// Mitsubishi GX Works2 project: GoodAfterChanges   PLC: FX3G

// global labels: Global1
VAR_GLOBAL
  Start_Day AT X007 : BOOL;
  Output_Analog AT D8282 : INT;
  Check_Input AT M1 : BOOL;
  Work_Day_Light AT Y007 : BOOL;
  End_Day AT M0 : BOOL;
END_VAR
VAR_GLOBAL CONSTANT
  Petel_For_Regular : REAL := 280;
  Lemon_For_Regular : REAL := 455;
END_VAR
VAR_GLOBAL
  Input_Petel AT D2000 : REAL;
  Input_Lemon AT D2002 : REAL;
  Input_Gummy_Bears AT D2004 : REAL;
  Input_Stabilizer AT D2006 : REAL;
  Stock_Petel AT D3000 : REAL;
  Stock_Lemon AT D3002 : REAL;
  Stock_Gummy_Bears AT D3004 : REAL;
  Stock_Stabilizer AT D3006 : REAL;
  Read_Input AT X001 : BOOL;
END_VAR
VAR_GLOBAL CONSTANT
  Petel_For_Special : REAL := 385;
  Lemon_For_Special : REAL := 665;
  Gummy_Bears_For_Special : REAL := 70;
  Stabilizer_For_Special : REAL := 30;
END_VAR
VAR_GLOBAL
  Input_Analog1 AT D8280 : INT;
END_VAR
VAR_GLOBAL CONSTANT
  Normalize : REAL := 404.5;
END_VAR
VAR_GLOBAL
  Type_Ice_Cream AT D4000 : REAL;
END_VAR
VAR_GLOBAL CONSTANT
  Min_Regular : REAL;
  Min_Special : REAL := 6;
  Max_Regular : REAL := 5.0;
END_VAR
VAR_GLOBAL
  Making_Ice_Cream AT Y000 : BOOL;
  Making_Time AT TC1 : BOOL;
  End_Making AT TS1 : BOOL;
  Start_Cooling AT X002 : BOOL;
  Petel_Making AT D4200 : REAL;
  Lemon_Making AT D4202 : REAL;
END_VAR
VAR_GLOBAL CONSTANT
  Total_Petel_Regular : REAL := 350;
  Total_Petel_Special : REAL := 560;
  Total_Lemon_Regular : REAL := 490;
  Total_Lemon_Special : REAL := 700;
END_VAR
VAR_GLOBAL
  Petel_Cooling AT D4204 : REAL;
  Cool_Time AT TC2 : BOOL;
END_VAR
VAR_GLOBAL CONSTANT
  Time_Making_Sec : WORD := 50;
  Time_Cool_Sec : WORD := 80;
END_VAR
VAR_GLOBAL
  Mixing_Pot AT D4208 : REAL;
  Mixing_Reg_Time AT TC3 : BOOL;
  Mixing_Spe_Time AT TC4 : BOOL;
END_VAR
VAR_GLOBAL CONSTANT
  Mixing_Reg_Sec : WORD := 30;
  Mixing_Spe_Sec : WORD := 50;
END_VAR
VAR_GLOBAL
  Regular_Check AT M3 : BOOL;
  Special_Check AT M4 : BOOL;
  Make_Special AT M6 : BOOL;
  Make_Regular AT M5 : BOOL;
  End_Cooling AT TS2 : BOOL;
  Cooling_Ice_Cream AT Y002 : BOOL;
  Temp_Sensor AT X003 : BOOL;
  End_Regular_Mixing AT TS3 : BOOL;
  End_Special_Mixing AT TS4 : BOOL;
  Blink_Helper AT M7 : BOOL;
  Light5 AT Y005 : BOOL;
END_VAR
VAR_GLOBAL CONSTANT
  Blinking_Time : WORD := 5;
END_VAR
VAR_GLOBAL
  Start_Packing AT X004 : BOOL;
  First_Cup AT CC0 : BOOL;
END_VAR
VAR_GLOBAL CONSTANT
  Counter1 : WORD := 1;
END_VAR
VAR_GLOBAL
  Counter_Pack AT CC1 : BOOL;
END_VAR
VAR_GLOBAL CONSTANT
  Counter7 : WORD := 7;
END_VAR
VAR_GLOBAL
  End_Counter1 AT CS0 : BOOL;
  End_Counter7 AT CS1 : BOOL;
  Light4 AT Y004 : BOOL;
  Pack_One AT X000 : BOOL;
  Packs_Amount AT D4400 : REAL;
END_VAR
VAR_GLOBAL CONSTANT
  Add_One : REAL := 1;
END_VAR
VAR_GLOBAL
  Update_Stock AT M2 : BOOL;
END_VAR
VAR_GLOBAL CONSTANT
  Max_Special : REAL := 10.0;
  Gummy_Bears_For_Regular : REAL := 28;
  Stabilizer_For_Regular : REAL := 15;
END_VAR
VAR_GLOBAL
  Lemon_Cooling AT D4206 : REAL;
  Blink5 AT TC5 : BOOL;
  Blink6 AT TC6 : BOOL;
  End_Blink5 AT TS5 : BOOL;
  Light6 AT Y006 : BOOL;
  End_Blink6 AT TS6 : BOOL;
  Emergency_Stop AT X005 : BOOL;
  Finish_Reset AT M8 : BOOL;
END_VAR
VAR_GLOBAL CONSTANT
  Normalize_Back : REAL := 40.45;
END_VAR

// task Task_01 (event TRUE, interval 0, priority 31): POU_01

PROGRAM POU_01
(* structured ladder/FBD written out as ST: instructions are called as NAME(EN, inputs, outputs); _pN, _eN, _tN stand for wires *)
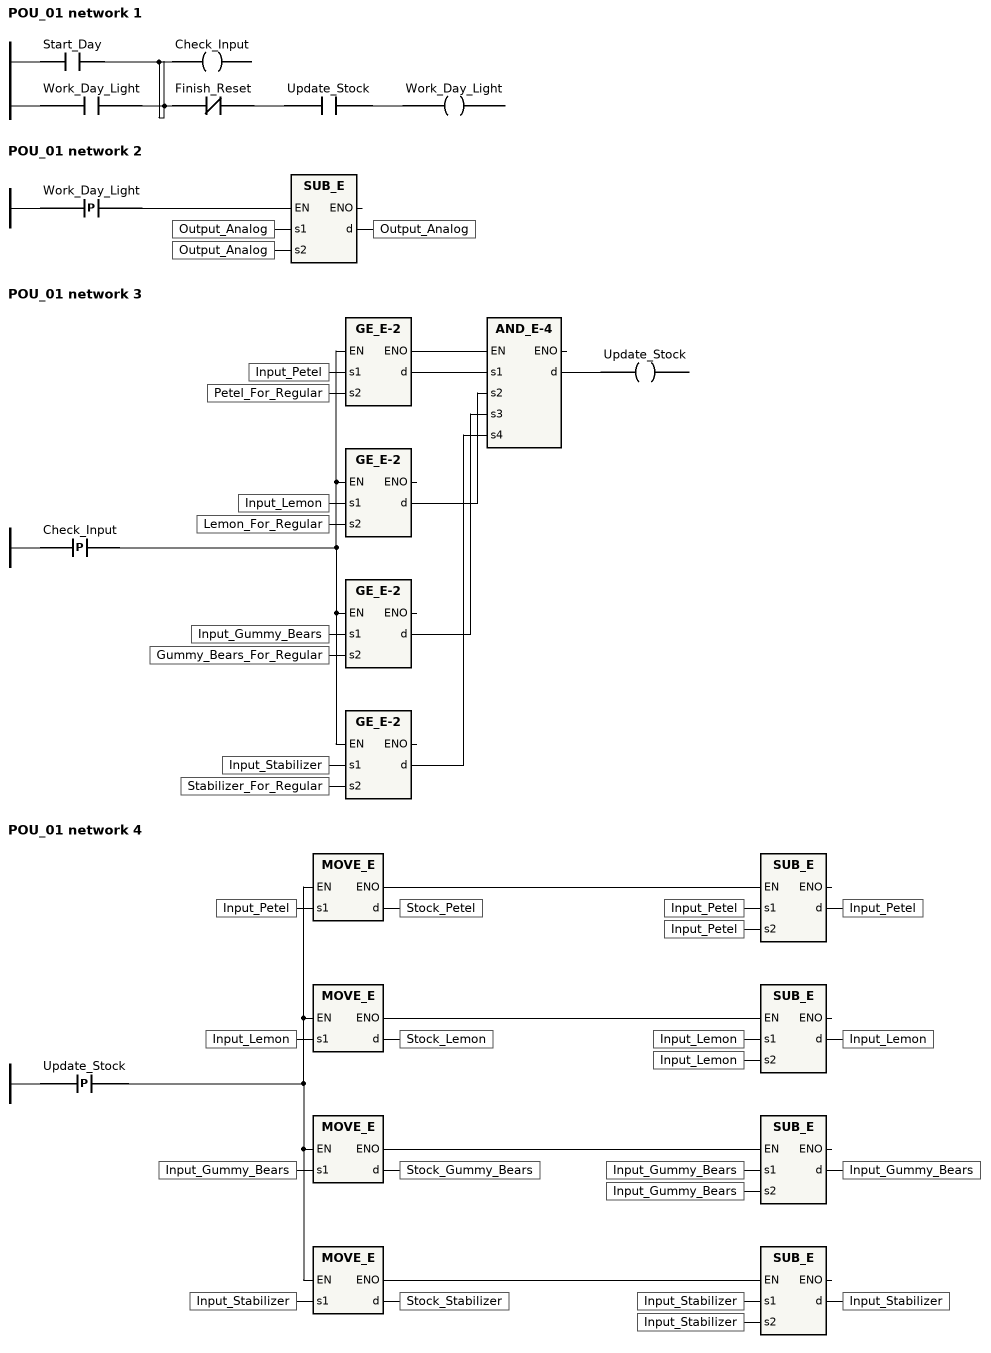
(* network 1 *)
_p1 := Start_Day OR Work_Day_Light;
Check_Input := _p1;
Work_Day_Light := _p1 AND NOT Finish_Reset AND Update_Stock;
(* network 2 *)
SUB_E(LDP(TRUE, Work_Day_Light), Output_Analog, Output_Analog, Output_Analog);
(* network 3 *)
_p1 := LDP(TRUE, Check_Input);
_e3 := GE_E(_p1, Input_Petel, Petel_For_Regular, _t2);
GE_E(_p1, Input_Lemon, Lemon_For_Regular, _t4);
GE_E(_p1, Input_Gummy_Bears, Gummy_Bears_For_Regular, _t5);
GE_E(_p1, Input_Stabilizer, Stabilizer_For_Regular, _t6);
AND_E(_e3, _t2, _t4, _t5, _t6, _t7);
Update_Stock := _t7;
(* network 4 *)
_p1 := LDP(TRUE, Update_Stock);
_e2 := MOVE_E(_p1, Input_Petel, Stock_Petel);
SUB_E(_e2, Input_Petel, Input_Petel, Input_Petel);
_e3 := MOVE_E(_p1, Input_Lemon, Stock_Lemon);
SUB_E(_e3, Input_Lemon, Input_Lemon, Input_Lemon);
_e4 := MOVE_E(_p1, Input_Gummy_Bears, Stock_Gummy_Bears);
SUB_E(_e4, Input_Gummy_Bears, Input_Gummy_Bears, Input_Gummy_Bears);
_e5 := MOVE_E(_p1, Input_Stabilizer, Stock_Stabilizer);
SUB_E(_e5, Input_Stabilizer, Input_Stabilizer, Input_Stabilizer);
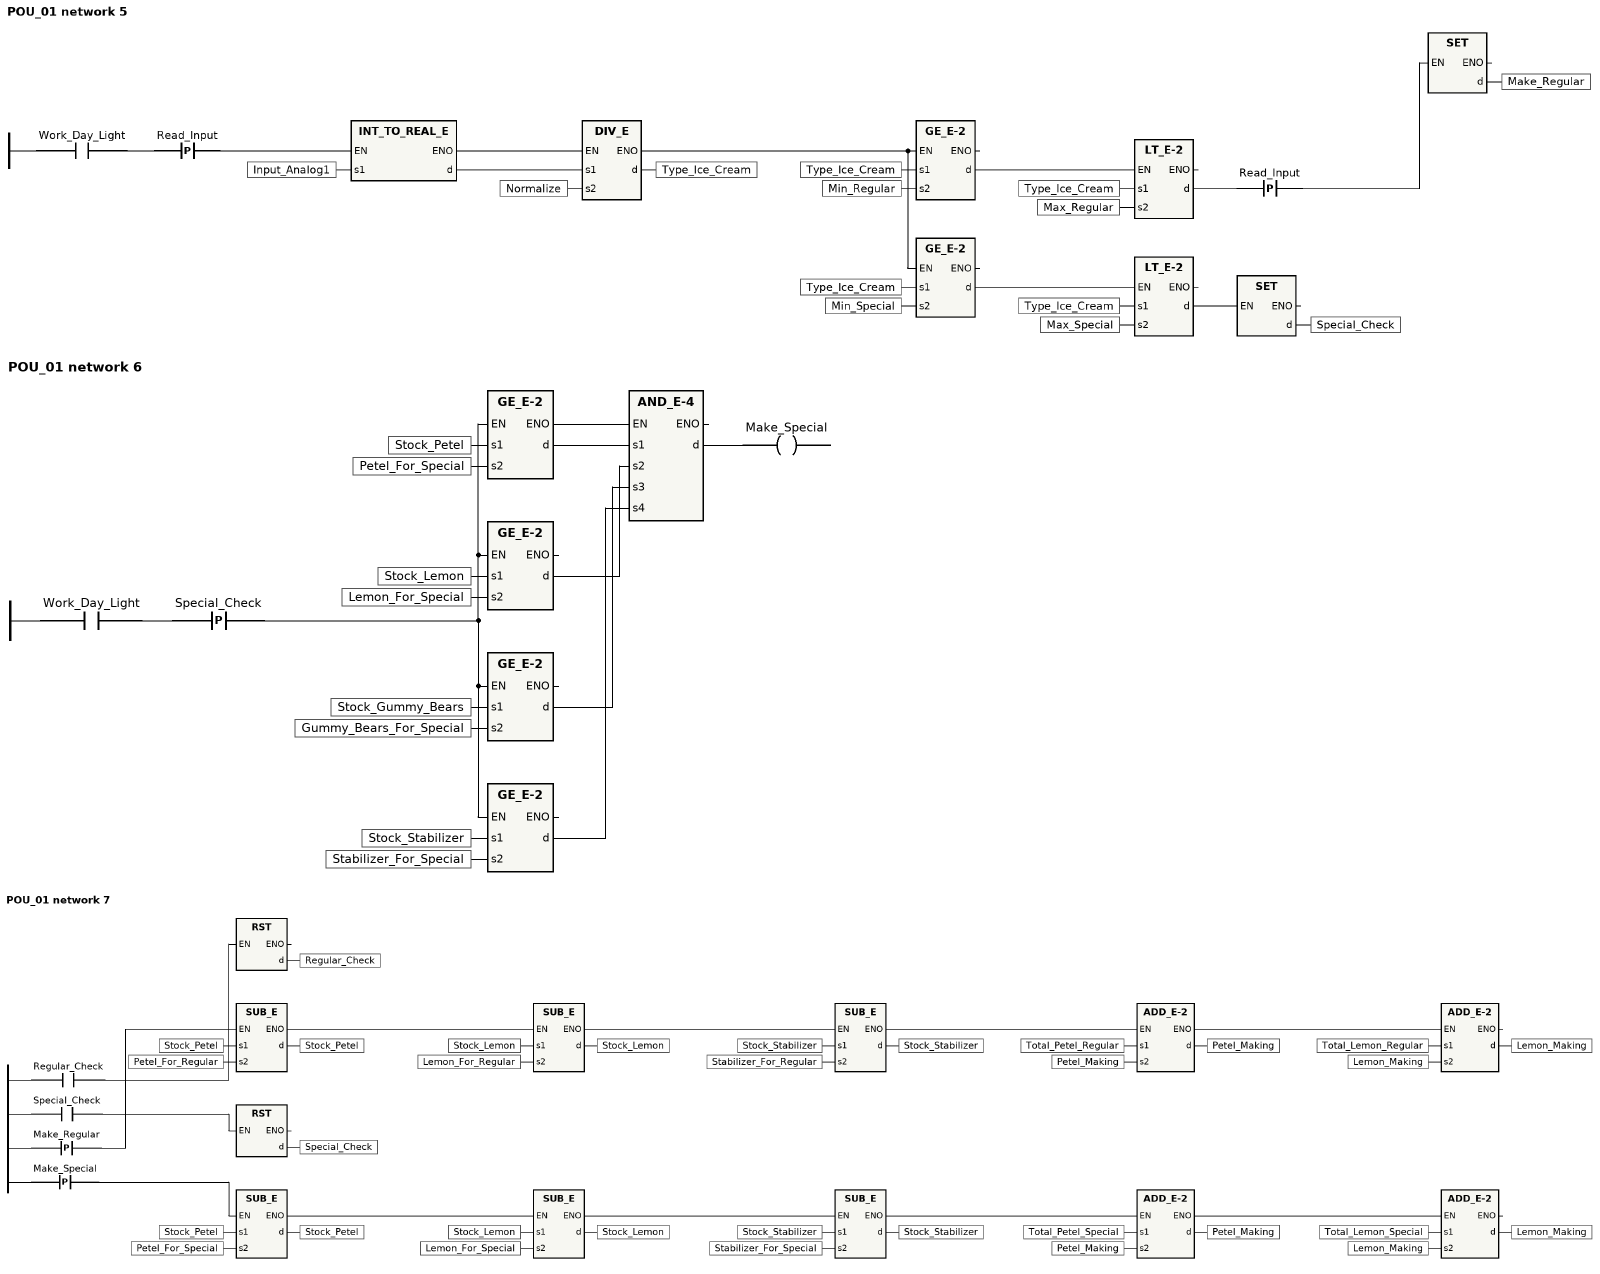
(* network 5 *)
_e2 := INT_TO_REAL_E(Work_Day_Light AND LDP(TRUE, Read_Input), Input_Analog1, _t1);
_e3 := DIV_E(_e2, _t1, Normalize, Type_Ice_Cream);
GE_E(_e3, Type_Ice_Cream, Min_Regular, _t4);
LT_E(_t4, Type_Ice_Cream, Max_Regular, _t5);
SET(_t5 AND LDP(TRUE, Read_Input), Make_Regular);
GE_E(_e3, Type_Ice_Cream, Min_Special, _t6);
LT_E(_t6, Type_Ice_Cream, Max_Special, _t7);
SET(_t7, Special_Check);
(* network 6 *)
_p1 := Work_Day_Light AND LDP(TRUE, Special_Check);
_e3 := GE_E(_p1, Stock_Petel, Petel_For_Special, _t2);
GE_E(_p1, Stock_Lemon, Lemon_For_Special, _t4);
GE_E(_p1, Stock_Gummy_Bears, Gummy_Bears_For_Special, _t5);
GE_E(_p1, Stock_Stabilizer, Stabilizer_For_Special, _t6);
AND_E(_e3, _t2, _t4, _t5, _t6, _t7);
Make_Special := _t7;
(* network 7 *)
RST(Regular_Check, Regular_Check);
RST(Special_Check, Special_Check);
_e1 := SUB_E(LDP(TRUE, Make_Regular), Stock_Petel, Petel_For_Regular, Stock_Petel);
_e2 := SUB_E(_e1, Stock_Lemon, Lemon_For_Regular, Stock_Lemon);
_e3 := SUB_E(_e2, Stock_Stabilizer, Stabilizer_For_Regular, Stock_Stabilizer);
_e4 := ADD_E(_e3, Total_Petel_Regular, Petel_Making, Petel_Making);
ADD_E(_e4, Total_Lemon_Regular, Lemon_Making, Lemon_Making);
_e5 := SUB_E(LDP(TRUE, Make_Special), Stock_Petel, Petel_For_Special, Stock_Petel);
_e6 := SUB_E(_e5, Stock_Lemon, Lemon_For_Special, Stock_Lemon);
_e7 := SUB_E(_e6, Stock_Stabilizer, Stabilizer_For_Special, Stock_Stabilizer);
_e8 := ADD_E(_e7, Total_Petel_Special, Petel_Making, Petel_Making);
ADD_E(_e8, Total_Lemon_Special, Lemon_Making, Lemon_Making);
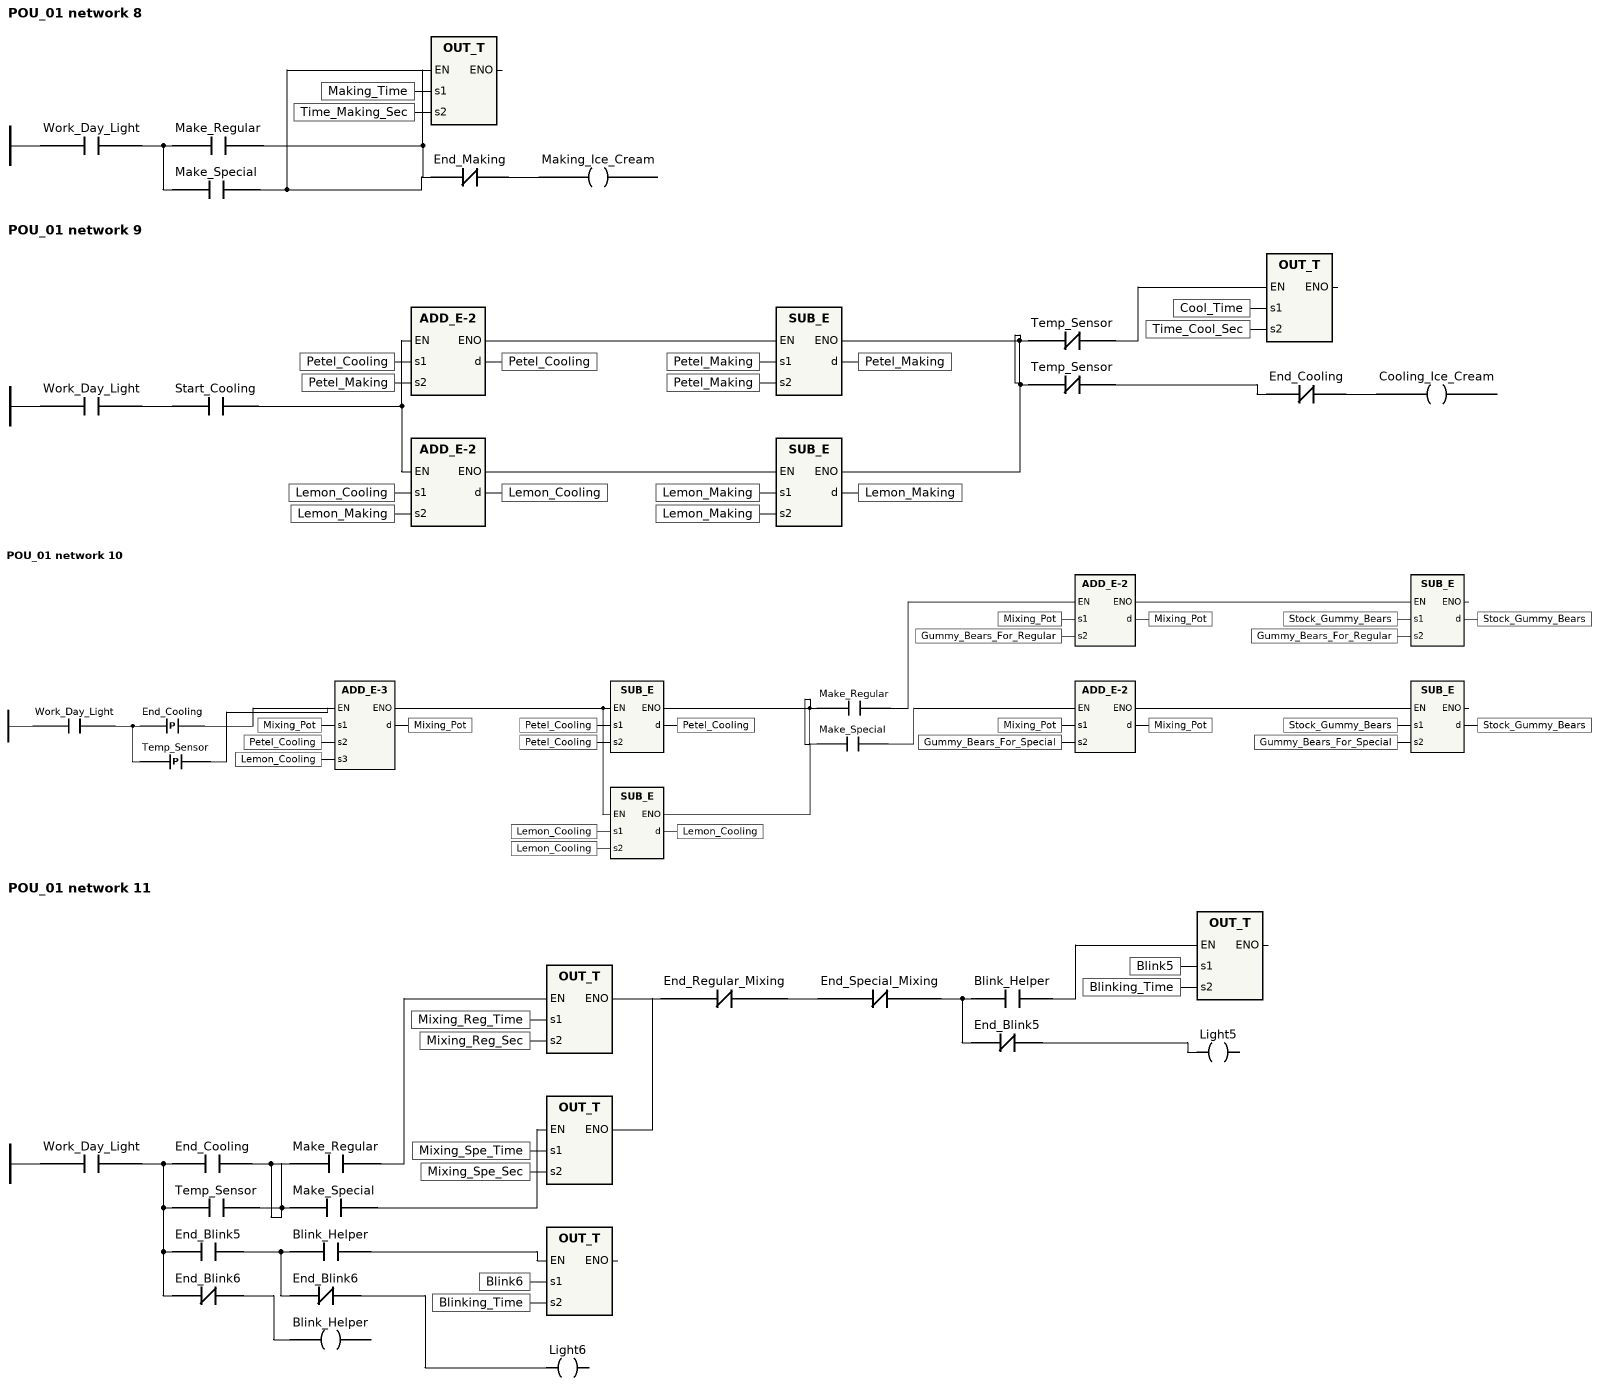
(* network 8 *)
_p1 := (Work_Day_Light AND Make_Regular) OR (Work_Day_Light AND Make_Special);
OUT_T(_p1, Making_Time, Time_Making_Sec);
Making_Ice_Cream := _p1 AND NOT End_Making;
(* network 9 *)
_p1 := Work_Day_Light AND Start_Cooling;
_e2 := ADD_E(_p1, Petel_Cooling, Petel_Making, Petel_Cooling);
_e3 := SUB_E(_e2, Petel_Making, Petel_Making, Petel_Making);
_e4 := ADD_E(_p1, Lemon_Cooling, Lemon_Making, Lemon_Cooling);
_e5 := SUB_E(_e4, Lemon_Making, Lemon_Making, Lemon_Making);
_p6 := _e3 OR _e5;
OUT_T(_p6 AND NOT Temp_Sensor, Cool_Time, Time_Cool_Sec);
Cooling_Ice_Cream := _p6 AND NOT Temp_Sensor AND NOT End_Cooling;
(* network 10 *)
_e1 := ADD_E((Work_Day_Light AND LDP(TRUE, End_Cooling)) OR (Work_Day_Light AND LDP(TRUE, Temp_Sensor)), Mixing_Pot, Petel_Cooling, Lemon_Cooling, Mixing_Pot);
_e2 := SUB_E(_e1, Petel_Cooling, Petel_Cooling, Petel_Cooling);
_e3 := SUB_E(_e1, Lemon_Cooling, Lemon_Cooling, Lemon_Cooling);
_p4 := _e2 OR _e3;
_e5 := ADD_E(_p4 AND Make_Regular, Mixing_Pot, Gummy_Bears_For_Regular, Mixing_Pot);
SUB_E(_e5, Stock_Gummy_Bears, Gummy_Bears_For_Regular, Stock_Gummy_Bears);
_e6 := ADD_E(_p4 AND Make_Special, Mixing_Pot, Gummy_Bears_For_Special, Mixing_Pot);
SUB_E(_e6, Stock_Gummy_Bears, Gummy_Bears_For_Special, Stock_Gummy_Bears);
(* network 11 *)
_p1 := (Work_Day_Light AND End_Cooling) OR (Work_Day_Light AND Temp_Sensor);
_e2 := OUT_T(_p1 AND Make_Regular, Mixing_Reg_Time, Mixing_Reg_Sec);
_e3 := OUT_T(_p1 AND Make_Special, Mixing_Spe_Time, Mixing_Spe_Sec);
_p4 := ((_e2 OR _e3) AND NOT End_Regular_Mixing) AND NOT End_Special_Mixing;
OUT_T(_p4 AND Blink_Helper, Blink5, Blinking_Time);
Light5 := _p4 AND NOT End_Blink5;
_p5 := Work_Day_Light AND End_Blink5;
OUT_T(_p5 AND Blink_Helper, Blink6, Blinking_Time);
Light6 := _p5 AND NOT End_Blink6;
Blink_Helper := Work_Day_Light AND NOT End_Blink6;
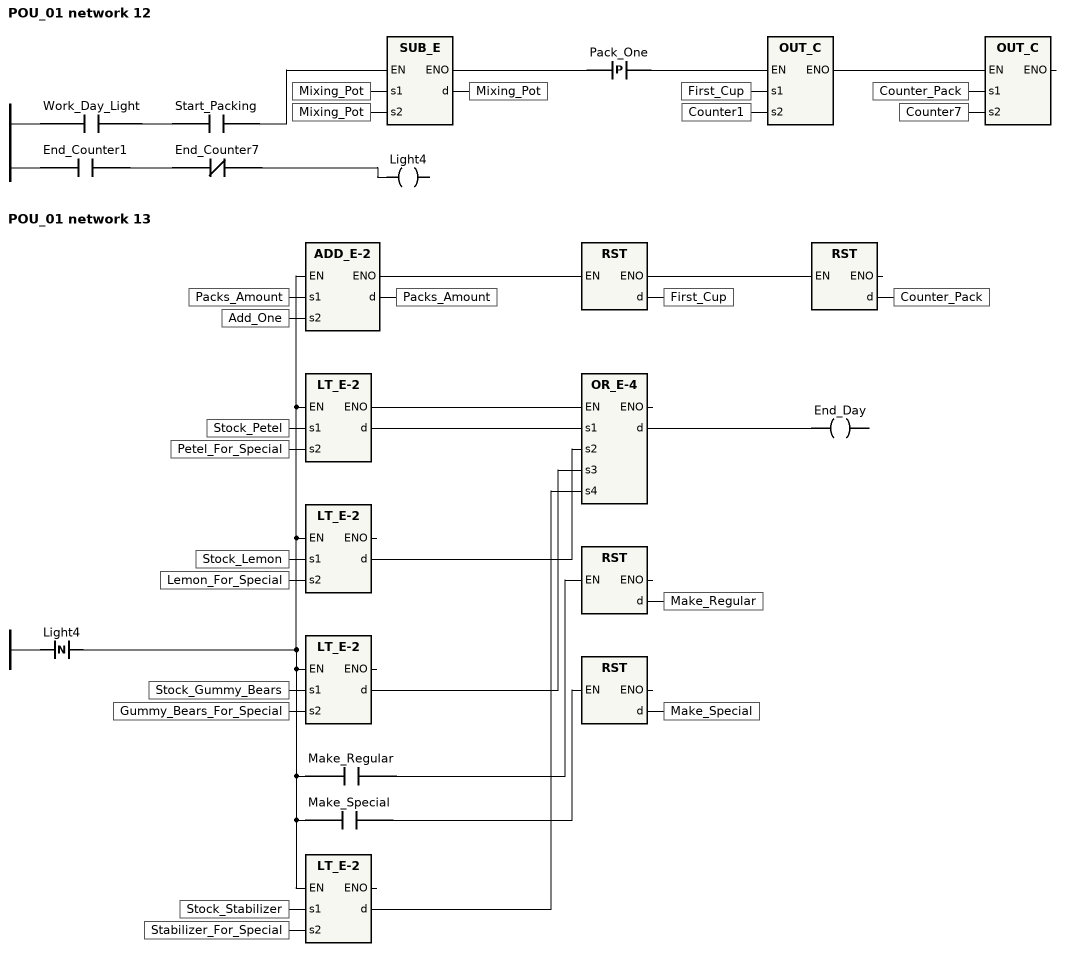
(* network 12 *)
_e1 := SUB_E(Work_Day_Light AND Start_Packing, Mixing_Pot, Mixing_Pot, Mixing_Pot);
_e2 := OUT_C(_e1 AND LDP(TRUE, Pack_One), First_Cup, Counter1);
OUT_C(_e2, Counter_Pack, Counter7);
Light4 := End_Counter1 AND NOT End_Counter7;
(* network 13 *)
_p1 := LDF(TRUE, Light4);
_e2 := ADD_E(_p1, Packs_Amount, Add_One, Packs_Amount);
_e3 := RST(_e2, First_Cup);
RST(_e3, Counter_Pack);
RST(_p1 AND Make_Regular, Make_Regular);
_e5 := LT_E(_p1, Stock_Petel, Petel_For_Special, _t4);
RST(_p1 AND Make_Special, Make_Special);
LT_E(_p1, Stock_Lemon, Lemon_For_Special, _t6);
LT_E(_p1, Stock_Gummy_Bears, Gummy_Bears_For_Special, _t7);
LT_E(_p1, Stock_Stabilizer, Stabilizer_For_Special, _t8);
OR_E(_e5, _t4, _t6, _t7, _t8, _t9);
End_Day := _t9;
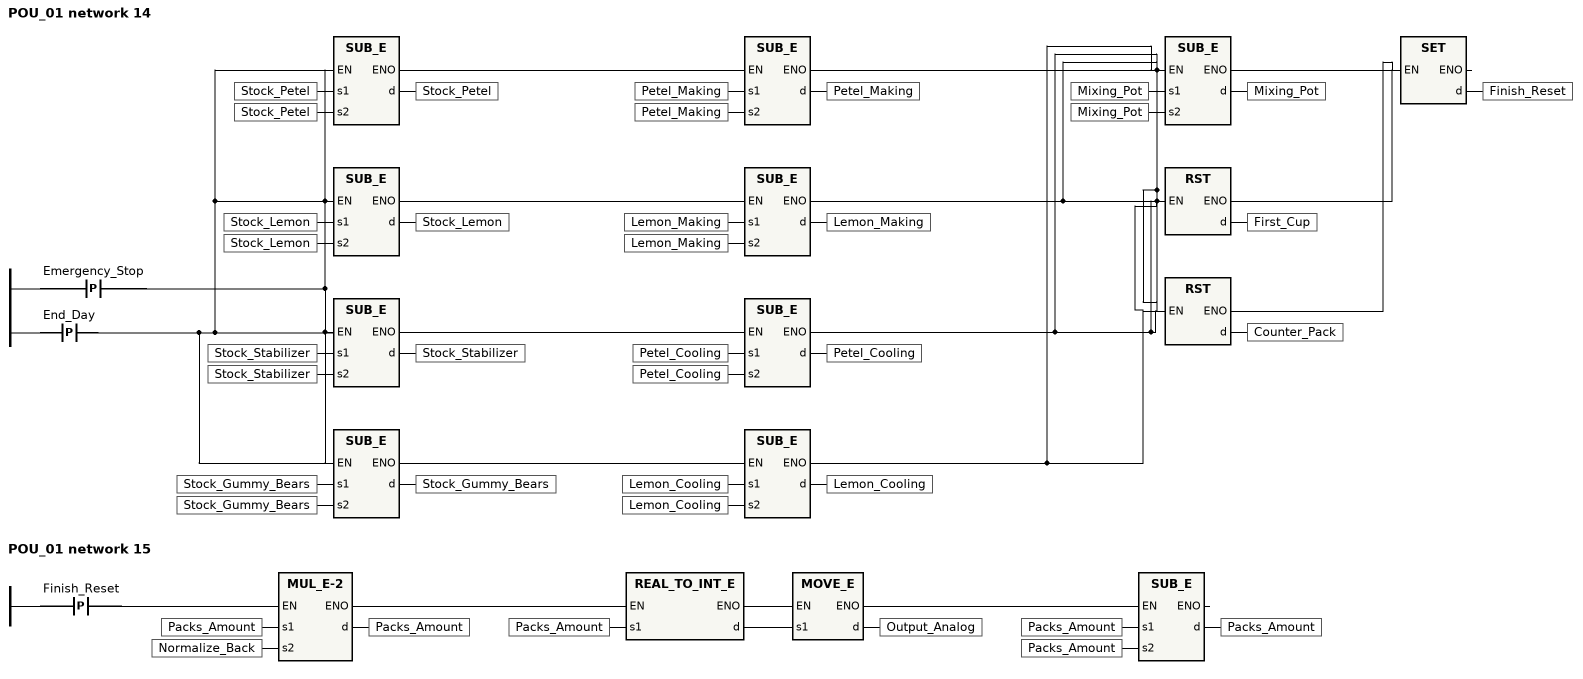
(* network 14 *)
_p1 := LDP(TRUE, Emergency_Stop) OR LDP(TRUE, End_Day);
_e2 := SUB_E(_p1, Stock_Petel, Stock_Petel, Stock_Petel);
_e3 := SUB_E(_e2, Petel_Making, Petel_Making, Petel_Making);
_e4 := SUB_E(_p1, Stock_Lemon, Stock_Lemon, Stock_Lemon);
_e5 := SUB_E(_e4, Lemon_Making, Lemon_Making, Lemon_Making);
_e6 := SUB_E(_p1, Stock_Stabilizer, Stock_Stabilizer, Stock_Stabilizer);
_e7 := SUB_E(_e6, Petel_Cooling, Petel_Cooling, Petel_Cooling);
_e8 := SUB_E(_p1, Stock_Gummy_Bears, Stock_Gummy_Bears, Stock_Gummy_Bears);
_e9 := SUB_E(_e8, Lemon_Cooling, Lemon_Cooling, Lemon_Cooling);
_p10 := _e3 OR _e5 OR _e7 OR _e9;
_e11 := SUB_E(_p10, Mixing_Pot, Mixing_Pot, Mixing_Pot);
_e12 := RST(_p10, First_Cup);
_e13 := RST(_p10, Counter_Pack);
SET(_e11 OR _e12 OR _e13, Finish_Reset);
(* network 15 *)
_e1 := MUL_E(LDP(TRUE, Finish_Reset), Packs_Amount, Normalize_Back, Packs_Amount);
_e3 := REAL_TO_INT_E(_e1, Packs_Amount, _t2);
_e4 := MOVE_E(_e3, _t2, Output_Analog);
SUB_E(_e4, Packs_Amount, Packs_Amount, Packs_Amount);
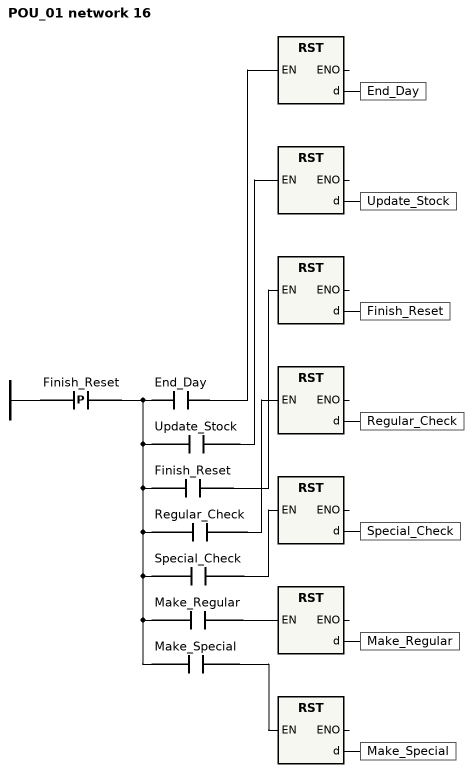
(* network 16 *)
_p1 := LDP(TRUE, Finish_Reset);
RST(_p1 AND End_Day, End_Day);
RST(_p1 AND Update_Stock, Update_Stock);
RST(_p1 AND Finish_Reset, Finish_Reset);
RST(_p1 AND Regular_Check, Regular_Check);
RST(_p1 AND Special_Check, Special_Check);
RST(_p1 AND Make_Regular, Make_Regular);
RST(_p1 AND Make_Special, Make_Special);
END_PROGRAM
